PROGRAM MAIN
VAR
//aProductArray : ARRAY[1..20] OF REAL := [23,120,85,100,250,489.95,489.96,230,190,30,10,600,240,210,10000,8600,61,349.444,42.252,534.2];
aProductArray : ARRAY[1..20] OF REAL;
stProductAnalysis : ST_ProductStats;
	bRun: BOOL:= TRUE;
	nBase : INT ;
END_VAR

IF bRun THEN
	RandomArrayGenerator(aProductArray,nBase);
	stProductAnalysis := AnalyzeBatch(aProductArray);
	//bRun := FALSE;
END_IF

END_PROGRAM

(* stored: Version 1.1.0.1, ProductVersion 3.1.4024.16
   POU MAIN: Id {864c6c48-a6ed-4662-b6a7-4e5a364ffb3e}, SpecialFunc None *)
